(* PLC project Unnamed, Unknown Unnamed 1 *)
(* stored: creationDateTime 2025-06-21T16:36:35, modificationDateTime 2025-06-21T17:39:55 *)

PROGRAM sema_pou
  VAR
    input1 AT %IX100.0 : BOOL;
    input2 AT %IX100.1 : BOOL;
    reset AT %IX100.2 : BOOL;
    load AT %IX100.3 : BOOL;
    output1 AT %QX100.0 : BOOL;
    output2 AT %QX100.1 : BOOL;
  END_VAR
  VAR
    SEMA0 : SEMA;
    RS0 : RS;
  END_VAR

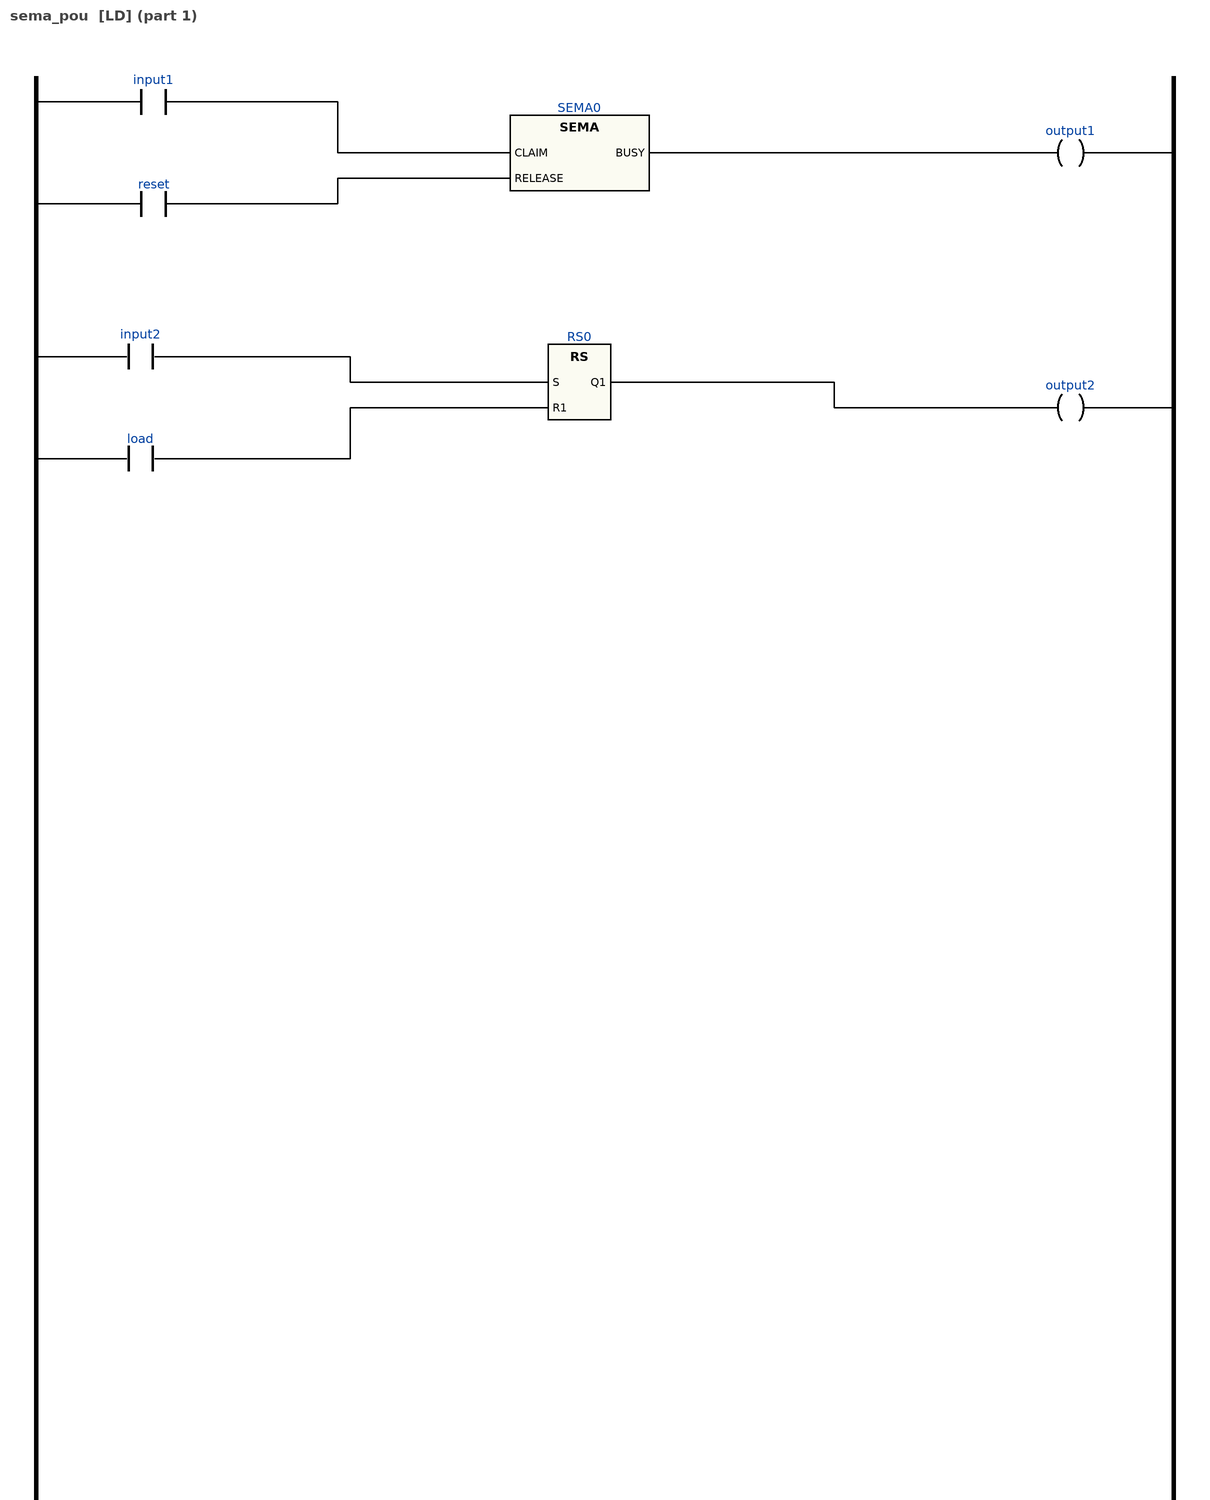
(* LD diagram, written out as Structured Text *)
SEMA0(CLAIM := input1, RELEASE := reset);
output1 := SEMA0.BUSY;
RS0(S := input2, R1 := load);
output2 := RS0.Q1;
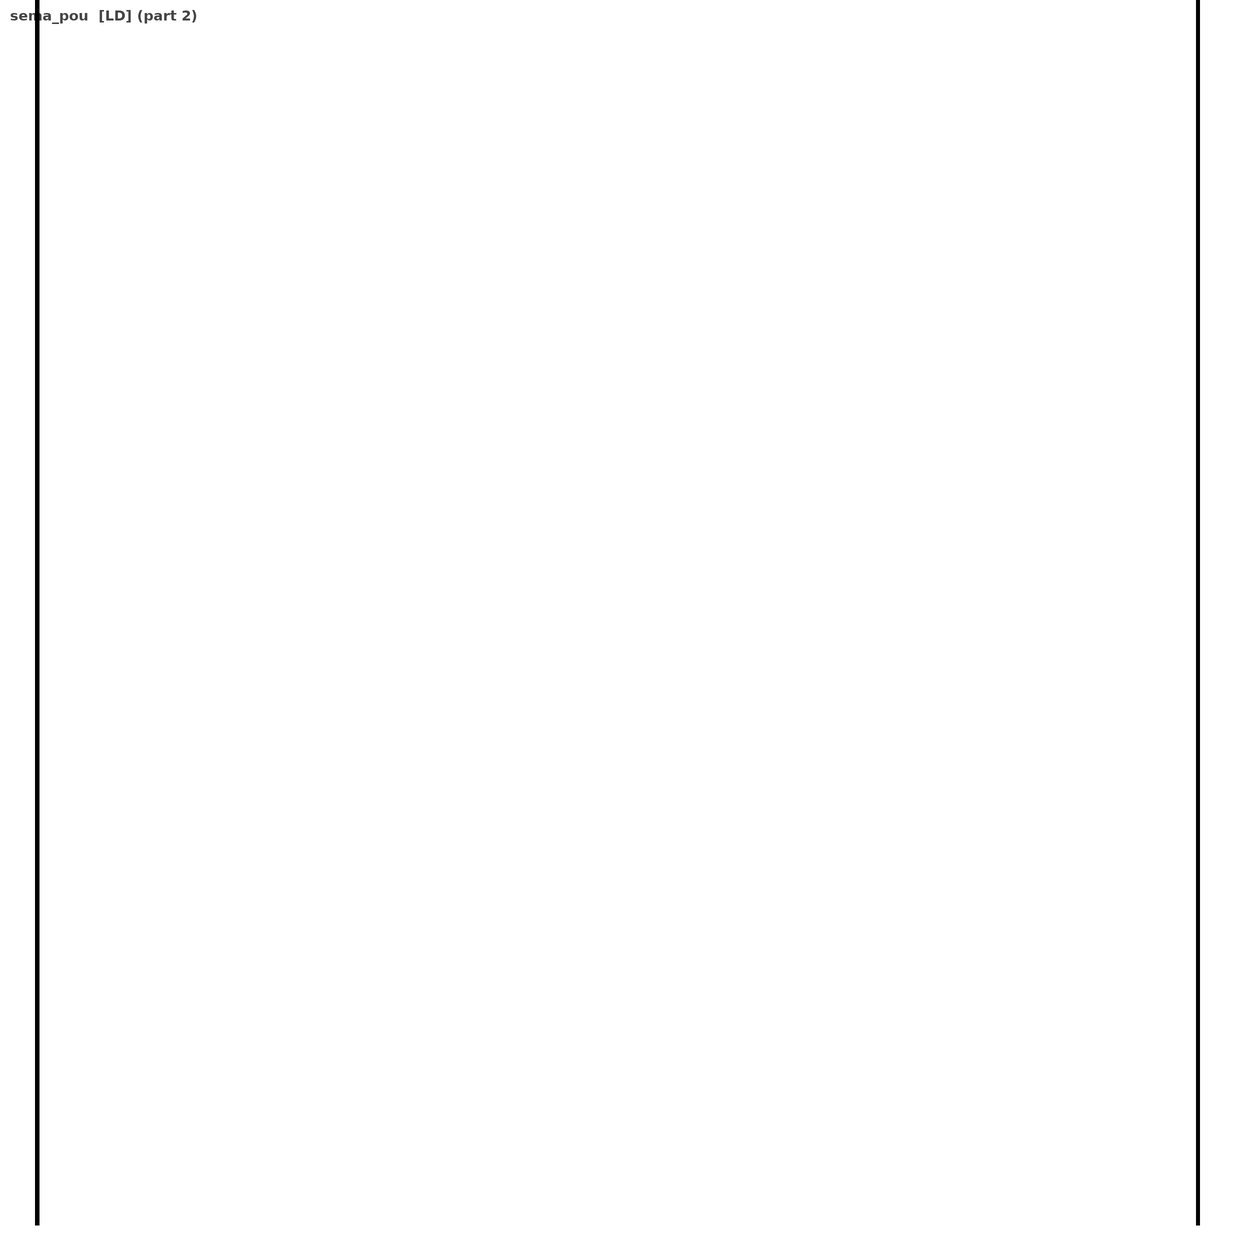
END_PROGRAM

CONFIGURATION Config0
  RESOURCE Res0 ON PLC
    TASK task0(INTERVAL := T#20ms, PRIORITY := 0);
    PROGRAM instance0 WITH task0 : sema_pou;
  END_RESOURCE
END_CONFIGURATION
